FUNCTION_BLOCK FB_PSp_Input
VAR_INPUT
	IN_Temp_oben	: REAL;
	IN_Temp_mitte	: REAL;
	IN_Temp_unten	: REAL;
END_VAR
VAR_OUTPUT
	Temp_oben		: REAL;
	Temp_mitte		: REAL;
	Temp_unten		: REAL;
END_VAR
VAR
END_VAR

Temp_oben		:= IN_Temp_oben;
Temp_mitte		:= IN_Temp_mitte;
Temp_unten		:= IN_Temp_unten;

END_FUNCTION_BLOCK

(* stored: Version 1.1.0.1, ProductVersion 3.1.4024.9
   POU FB_PSp_Input: Id {47d1b150-8f6b-4da0-a9ce-9024286d148d}, SpecialFunc None *)
